FUNCTION_BLOCK "MOTOR_CONTROL"
{ S7_Optimized_Access := 'TRUE' }
AUTHOR : TAI_NW
VERSION : 0.1
TITLE = Motor Control

VAR_INPUT
    Start : Bool;
    Stop  : Bool;
    timer : Time;
END_VAR

BEGIN
NETWORK
// Dit is een test
TITLE = INIT
    L 254;
    T #t_MaxWaardeVoorOverflow;
    ITD;
    T #t_MaxWaardeOverflowDINT;

    L  1000
    ITD
    DTR
    T #RealValue
END_FUNCTION_BLOCK